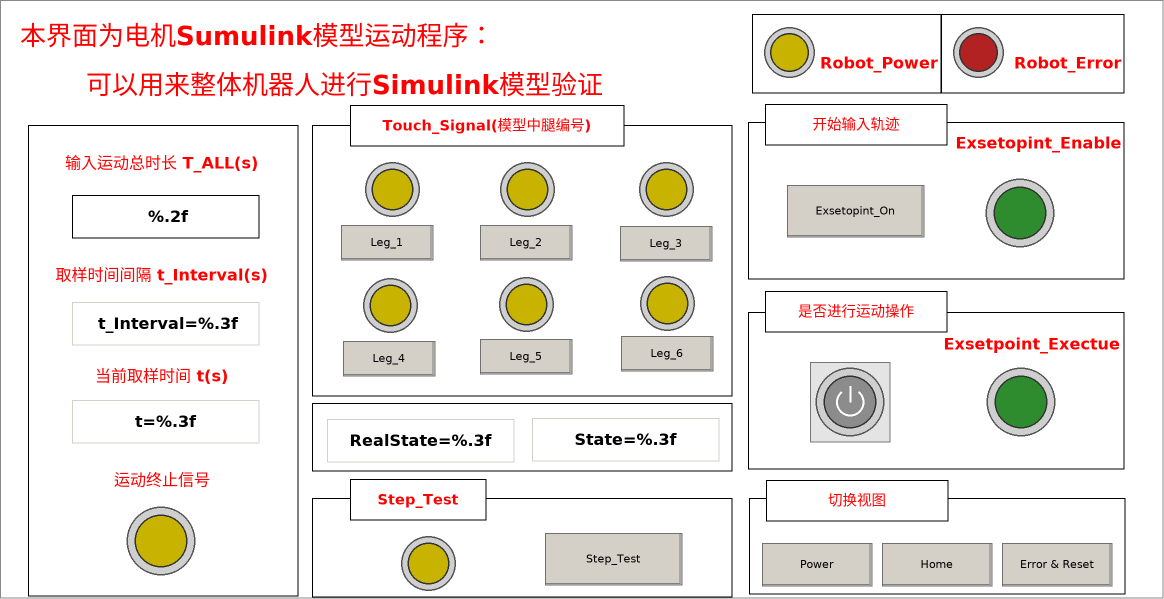
VISUALIZATION Visu_Walking_Robot_SimulinkMove  // 1164x599
    Rectangle (312,498 420x99)
    Rectangle (749,498 376x96)
    Rectangle (766,480 182x41), "切换视图"
    Button (762,543 110x43), "Power"
        OnMouseClick: change screen: Visu_Walking_Robot_Power
    Button (1002,543 110x43), "Error & Reset"
        OnMouseClick: change screen: Visu_Walking_Robot_Reset
    Button (882,543 110x43), "Home"
        OnMouseClick: change screen: Visu_Walking_Robot_Home
    Rectangle (28,125 270x471)
    Rectangle (752,14 189x79)
    Rectangle (748,312 376x157)
    Label (902,328 260x32), "Exsetpoint_Exectue"
    Rectangle (765,291 182x41), "是否进行运动操作"
    Lamp1 (981,362 80x80), variable: Walking_Robot_Movement.ExSetPoint_Execute, style: Lamp-Lamp1-Green
    PowerSwitch (810,362 80x80), variable: Walking_Robot_Movement.ExSetPoint_Execute, behaviour: TOGGLE, style: Switch-PowerSwitch-Gray
    Rectangle (941,14 183x79)
    Lamp1 (948,23 61x59), variable: Walking_Robot_Control.Robot_Error, style: Lamp-Lamp1-Red
    Label (991,47 154x32), "Robot_Error"
    Label (17,15 572x42), "本界面为电机Sumulink模型运动程序："
    Label (83,64 874x42), "可以用来整体机器人进行Simulink模型验证"
    Lamp1 (759,23 61x59), variable: Walking_Robot_Control.Robot_Power, style: Lamp-Lamp1-Yellow
    Label (802,47 154x32), "Robot_Power"
    Rectangle (748,122 376x157)
    Rectangle (765,104 182x41), "开始输入轨迹"
    Lamp1 (980,173 80x80), variable: Walking_Robot_Movement.ExtSetPointEnable, style: Lamp-Lamp1-Green
    Label (935,127 207x32), "Exsetopint_Enable"
    Rectangle (72,195 187x43), "%.2f", text variable: Walking_Robot_Movement.T_All
        OnMouseClick: write Walking_Robot_Movement.T_ALL via Default
    Label (32,147 260x32), "输入运动总时长 T_ALL(s)"
    Textfield (72,400 187x43), "t=%.3f", text variable: Walking_Robot_Movement.t
    Label (32,360 260x32), "当前取样时间 t(s)"
    Button (787,185 137x52), "Exsetopint_On"
        toggle Walking_Robot_Movement.ExtSetPointEnable
    Lamp1 (121,501 80x80), variable: Walking_Robot_Movement.ExtSetPointDisable, style: Lamp-Lamp1-Yellow
    Label (32,464 260x32), "运动终止信号"
    Label (32,259 260x32), "取样时间间隔 t_Interval(s)"
    Textfield (72,302 187x43), "t_Interval=%.3f", text variable: Walking_Robot_Movement.t_Interval
        OnMouseClick: write Walking_Robot_Movement.t_Interval via Default
    Rectangle (312,125 420x271)
    Rectangle (350,105 274x41), "Touch_Signal(模型中腿编号)"
    Lamp1 (361,157 63x65), variable: Walking_Robot_Movement.Touch_Signal[1], style: Lamp-Lamp1-Yellow
    Lamp1 (496,157 63x65), variable: Walking_Robot_Movement.Touch_Signal[2], style: Lamp-Lamp1-Yellow
    Lamp1 (635,157 63x65), variable: Walking_Robot_Movement.Touch_Signal[3], style: Lamp-Lamp1-Yellow
    Lamp1 (359,273 63x65), variable: Walking_Robot_Movement.Touch_Signal[4], style: Lamp-Lamp1-Yellow
    Lamp1 (495,272 63x65), variable: Walking_Robot_Movement.Touch_Signal[5], style: Lamp-Lamp1-Yellow
    Lamp1 (636,271 63x65), variable: Walking_Robot_Movement.Touch_Signal[6], style: Lamp-Lamp1-Yellow
    Rectangle (312,403 420x68)
    Textfield (327,419 187x43), "RealState=%.3f", text variable: Walking_Robot_Movement.realState
    Textfield (532,418 187x43), "State=%.3f", text variable: Walking_Robot_Movement.state
    Button (545,533 137x52), "Step_Test"
        toggle Walking_Robot_Movement.Step_Test
    Lamp1 (397,531 63x65), variable: Walking_Robot_Movement.Step_Test, style: Lamp-Lamp1-Yellow
    Rectangle (350,479 136x41), "Step_Test"
    Button (341,225 92x35), "Leg_1"
        toggle Walking_Robot_Movement.Touch_Signal[1]
    Button (480,225 92x35), "Leg_2"
        toggle Walking_Robot_Movement.Touch_Signal[2]
    Button (620,226 92x35), "Leg_3"
        toggle Walking_Robot_Movement.Touch_Signal[3]
    Button (343,341 92x35), "Leg_4"
        toggle Walking_Robot_Movement.Touch_Signal[4]
    Button (480,339 92x35), "Leg_5"
        toggle Walking_Robot_Movement.Touch_Signal[5]
    Button (621,336 92x35), "Leg_6"
        toggle Walking_Robot_Movement.Touch_Signal[6]
END_VISUALIZATION

(* stored: Version 1.1.0.1, ProductVersion 3.1.4020.12
   Visu Visu_Walking_Robot_SimulinkMove: Id {4953c662-5946-414d-97eb-1dec552a9040} *)
